# EPICS autosave request: iocBoot/iocTune/auto_settings_tuneSI.req
file "tune_settings.req",                  P=$(P),  R=$(R)
file "tuneSI_settings.req",                P=$(P),  R=$(R)
